FUNCTION_BLOCK FB_Tuer
VAR_INPUT
	SensorOpen1 : BOOL;
	SensorOpen2 : BOOL;
	SensorOpen3 : BOOL;
	SensorOpen4 : BOOL;
	SensorOpen5 : BOOL;
	SensorOpen6 : BOOL;
	
	SensorClosed1 : BOOL;
	SensorClosed2 : BOOL;
	SensorClosed3 : BOOL;
	SensorClosed4 : BOOL;
	SensorClosed5 : BOOL;
	SensorClosed6 : BOOL;
	
	Lichtschranke1 : BOOL;
	Lichtschranke2 : BOOL;
	Lichtschranke3 : BOOL;
	Lichtschranke4 : BOOL;
	Lichtschranke5 : BOOL;
	Lichtschranke6 : BOOL;
END_VAR
VAR_OUTPUT
	MotorOpen1 : BOOL;
	MotorOpen2 : BOOL;
	MotorOpen3 : BOOL;
	MotorOpen4 : BOOL;
	MotorOpen5 : BOOL;
	MotorOpen6 : BOOL;
	
	MotorClose1 : BOOL;
	MotorClose2 : BOOL;
	MotorClose3 : BOOL;
	MotorClose4 : BOOL;
	MotorClose5 : BOOL;
	MotorClose6 : BOOL;
	Done : BOOL;
	AllDoorsClosed : BOOL;
END_VAR
VAR
	TuerzyklusStarten : BOOL;
	Stockwerk : INT;
	State : ENUM_Tuer;
	ton1 : TON;
	ton2 : TON;
	ton3 : TON;
	ton4 : TON;
	ton5 : TON;
	ton6 : TON;
	Tueroffen : BOOL;
	bCloseAllMode : BOOL;
END_VAR

Done := FALSE;
ton1(IN := State = ENUM_Tuer.TuereAuf AND SensorOpen1, PT := T#2S);
ton2(IN := State = ENUM_Tuer.TuereAuf AND SensorOpen2, PT := T#2S);
ton3(IN := State = ENUM_Tuer.TuereAuf AND SensorOpen3, PT := T#2S);
ton4(IN := State = ENUM_Tuer.TuereAuf AND SensorOpen4, PT := T#2S);
ton5(IN := State = ENUM_Tuer.TuereAuf AND SensorOpen5, PT := T#2S);
ton6(IN := State = ENUM_Tuer.TuereAuf AND SensorOpen6, PT := T#2S);
IF bCloseAllMode THEN
    // Alle Türen schliessen – normaler State-Machine wird überbrückt
    MotorOpen1 := FALSE;
    IF NOT Lichtschranke1 THEN
        MotorClose1 := FALSE;
    ELSIF NOT SensorClosed1 THEN
        MotorClose1 := TRUE;
    ELSE
        MotorClose1 := FALSE;
    END_IF
    MotorOpen2 := FALSE;
    IF NOT Lichtschranke2 THEN
        MotorClose2 := FALSE;
    ELSIF NOT SensorClosed2 THEN
        MotorClose2 := TRUE;
    ELSE
        MotorClose2 := FALSE;
    END_IF
    MotorOpen3 := FALSE;
    IF NOT Lichtschranke3 THEN
        MotorClose3 := FALSE;
    ELSIF NOT SensorClosed3 THEN
        MotorClose3 := TRUE;
    ELSE
        MotorClose3 := FALSE;
    END_IF
    MotorOpen4 := FALSE;
    IF NOT Lichtschranke4 THEN
        MotorClose4 := FALSE;
    ELSIF NOT SensorClosed4 THEN
        MotorClose4 := TRUE;
    ELSE
        MotorClose4 := FALSE;
    END_IF
    MotorOpen5 := FALSE;
    IF NOT Lichtschranke5 THEN
        MotorClose5 := FALSE;
    ELSIF NOT SensorClosed5 THEN
        MotorClose5 := TRUE;
    ELSE
        MotorClose5 := FALSE;
    END_IF
    MotorOpen6 := FALSE;
    IF NOT Lichtschranke6 THEN
        MotorClose6 := FALSE;
    ELSIF NOT SensorClosed6 THEN
        MotorClose6 := TRUE;
    ELSE
        MotorClose6 := FALSE;
    END_IF
    // Wenn alle zu: Modus beenden
    IF SensorClosed1 AND SensorClosed2 AND SensorClosed3
       AND SensorClosed4 AND SensorClosed5 AND SensorClosed6 THEN
        bCloseAllMode := FALSE;
        Done := TRUE;
    END_IF
ELSE
    // Normaler Betrieb: Ausgänge zurücksetzen, dann State-Machine
    MotorOpen1 := FALSE;
    MotorClose1 := FALSE;
    MotorOpen2 := FALSE;
    MotorClose2 := FALSE;
    MotorOpen3 := FALSE;
    MotorClose3 := FALSE;
    MotorOpen4 := FALSE;
    MotorClose4 := FALSE;
    MotorOpen5 := FALSE;
    MotorClose5 := FALSE;
    MotorOpen6 := FALSE;
    MotorClose6 := FALSE;
    CASE State OF
        ENUM_Tuer.TuereZu:
            IF TuerzyklusStarten AND Stockwerk = 1 THEN
                State := ENUM_Tuer.TuereOeffnen;
            END_IF
            IF TuerzyklusStarten AND Stockwerk = 2 THEN
                State := ENUM_Tuer.TuereOeffnen;
            END_IF
            IF TuerzyklusStarten AND Stockwerk = 3 THEN
                State := ENUM_Tuer.TuereOeffnen;
            END_IF
            IF TuerzyklusStarten AND Stockwerk = 4 THEN
                State := ENUM_Tuer.TuereOeffnen;
            END_IF
            IF TuerzyklusStarten AND Stockwerk = 5 THEN
                State := ENUM_Tuer.TuereOeffnen;
            END_IF
            IF TuerzyklusStarten AND Stockwerk = 6 THEN
                State := ENUM_Tuer.TuereOeffnen;
            END_IF
        ENUM_Tuer.TuereOeffnen:
            Tueroffen := TRUE;
            IF Stockwerk = 1 THEN
                IF NOT SensorOpen1 THEN
                    MotorOpen1 := TRUE;
                ELSE
                    MotorOpen1 := FALSE;
                    State := ENUM_Tuer.TuereAuf;
                END_IF
            END_IF
            IF Stockwerk = 2 THEN
                IF NOT SensorOpen2 THEN
                    MotorOpen2 := TRUE;
                ELSE
                    MotorOpen2 := FALSE;
                    State := ENUM_Tuer.TuereAuf;
                END_IF
            END_IF
            IF Stockwerk = 3 THEN
                IF NOT SensorOpen3 THEN
                    MotorOpen3 := TRUE;
                ELSE
                    MotorOpen3 := FALSE;
                    State := ENUM_Tuer.TuereAuf;
                END_IF
            END_IF
            IF Stockwerk = 4 THEN
                IF NOT SensorOpen4 THEN
                    MotorOpen4 := TRUE;
                ELSE
                    MotorOpen4 := FALSE;
                    State := ENUM_Tuer.TuereAuf;
                END_IF
            END_IF
            IF Stockwerk = 5 THEN
                IF NOT SensorOpen5 THEN
                    MotorOpen5 := TRUE;
                ELSE
                    MotorOpen5 := FALSE;
                    State := ENUM_Tuer.TuereAuf;
                END_IF
            END_IF
            IF Stockwerk = 6 THEN
                IF NOT SensorOpen6 THEN
                    MotorOpen6 := TRUE;
                ELSE
                    MotorOpen6 := FALSE;
                    State := ENUM_Tuer.TuereAuf;
                END_IF
            END_IF
        ENUM_Tuer.TuereAuf:
            Tueroffen := FALSE;
            IF Stockwerk = 1 AND ton1.Q THEN
                State := ENUM_Tuer.TuereSchliessen;
            END_IF
            IF Stockwerk = 2 AND ton2.Q THEN
                State := ENUM_Tuer.TuereSchliessen;
            END_IF
            IF Stockwerk = 3 AND ton3.Q THEN
                State := ENUM_Tuer.TuereSchliessen;
            END_IF
            IF Stockwerk = 4 AND ton4.Q THEN
                State := ENUM_Tuer.TuereSchliessen;
            END_IF
            IF Stockwerk = 5 AND ton5.Q THEN
                State := ENUM_Tuer.TuereSchliessen;
            END_IF
            IF Stockwerk = 6 AND ton6.Q THEN
                State := ENUM_Tuer.TuereSchliessen;
            END_IF
        ENUM_Tuer.TuereSchliessen:
            IF Stockwerk = 1 THEN
                IF NOT Lichtschranke1 THEN
                    MotorClose1 := FALSE;
                    State := ENUM_Tuer.TuereOeffnen;
                ELSIF NOT SensorClosed1 THEN
                    MotorClose1 := TRUE;
                ELSE
                    MotorClose1 := FALSE;
                    TuerzyklusStarten := FALSE;
                    Done := TRUE;
                    State := ENUM_Tuer.TuereZu;
                END_IF
            END_IF
            IF Stockwerk = 2 THEN
                IF NOT Lichtschranke2 THEN
                    MotorClose2 := FALSE;
                    State := ENUM_Tuer.TuereOeffnen;
                ELSIF NOT SensorClosed2 THEN
                    MotorClose2 := TRUE;
                ELSE
                    MotorClose2 := FALSE;
                    TuerzyklusStarten := FALSE;
                    Done := TRUE;
                    State := ENUM_Tuer.TuereZu;
                END_IF
            END_IF
            IF Stockwerk = 3 THEN
                IF NOT Lichtschranke3 THEN
                    MotorClose3 := FALSE;
                    State := ENUM_Tuer.TuereOeffnen;
                ELSIF NOT SensorClosed3 THEN
                    MotorClose3 := TRUE;
                ELSE
                    MotorClose3 := FALSE;
                    TuerzyklusStarten := FALSE;
                    Done := TRUE;
                    State := ENUM_Tuer.TuereZu;
                END_IF
            END_IF
            IF Stockwerk = 4 THEN
                IF NOT Lichtschranke4 THEN
                    MotorClose4 := FALSE;
                    State := ENUM_Tuer.TuereOeffnen;
                ELSIF NOT SensorClosed4 THEN
                    MotorClose4 := TRUE;
                ELSE
                    MotorClose4 := FALSE;
                    TuerzyklusStarten := FALSE;
                    Done := TRUE;
                    State := ENUM_Tuer.TuereZu;
                END_IF
            END_IF
            IF Stockwerk = 5 THEN
                IF NOT Lichtschranke5 THEN
                    MotorClose5 := FALSE;
                    State := ENUM_Tuer.TuereOeffnen;
                ELSIF NOT SensorClosed5 THEN
                    MotorClose5 := TRUE;
                ELSE
                    MotorClose5 := FALSE;
                    TuerzyklusStarten := FALSE;
                    Done := TRUE;
                    State := ENUM_Tuer.TuereZu;
                END_IF
            END_IF
            IF Stockwerk = 6 THEN
                IF NOT Lichtschranke6 THEN
                    MotorClose6 := FALSE;
                    State := ENUM_Tuer.TuereOeffnen;
                ELSIF NOT SensorClosed6 THEN
                    MotorClose6 := TRUE;
                ELSE
                    MotorClose6 := FALSE;
                    TuerzyklusStarten := FALSE;
                    Done := TRUE;
                    State := ENUM_Tuer.TuereZu;
                END_IF
            END_IF
        ENUM_Tuer.Error:
    END_CASE
END_IF

IF IO_L1.Door_1_SensorClosed AND IO_L1.Door_2_SensorClosed AND IO_L1.Door_3_SensorClosed AND IO_L1.Door_4_SensorClosed AND IO_L1.Door_5_SensorClosed AND IO_L1.Door_6_SensorClosed THEN
	AllDoorsClosed := TRUE;
ELSE
	AllDoorsClosed := FALSE;
END_IF

METHOD PUBLIC M_AreDoorsClosed : BOOL
VAR_INPUT
END_VAR
IF IO_L1.Door_1_SensorClosed AND IO_L1.Door_2_SensorClosed AND IO_L1.Door_3_SensorClosed AND IO_L1.Door_4_SensorClosed AND IO_L1.Door_5_SensorClosed AND IO_L1.Door_6_SensorClosed THEN
	M_AreDoorsClosed := TRUE;
ELSE
	M_AreDoorsClosed := FALSE;
END_IF
END_METHOD

METHOD PUBLIC M_closeAllDoors : BOOL
VAR_INPUT
END_VAR
VAR
	Tuer1zu : BOOL;
	Tuer2zu : BOOL;
	Tuer3zu : BOOL;
	Tuer4zu : BOOL;
	Tuer5zu : BOOL;
	Tuer6zu : BOOL;
END_VAR

bCloseAllMode := TRUE;

M_closeAllDoors :=
    SensorClosed1 AND SensorClosed2 AND SensorClosed3 AND
    SensorClosed4 AND SensorClosed5 AND SensorClosed6;
END_METHOD

METHOD PUBLIC M_DoorOpen : BOOL
VAR_INPUT
	
END_VAR
IF Tueroffen THEN
	M_DoorOpen := TRUE;
ELSE
	M_DoorOpen := FALSE;
END_IF
END_METHOD

METHOD PUBLIC M_isDone : BOOL
VAR_INPUT
END_VAR
IF Done THEN
	M_isDone := TRUE;
ELSE 
	M_isDone := FALSE;
END_IF
END_METHOD

METHOD PUBLIC M_Tuerablaufstarten : BOOL
VAR_INPUT
	m_Stockwerk : INT;
END_VAR
IF m_Stockwerk >= 1 AND m_Stockwerk <= 6 THEN
	TuerzyklusStarten := TRUE;
	Stockwerk := m_Stockwerk;
	M_Tuerablaufstarten := TRUE;
ELSE
	M_Tuerablaufstarten := FALSE;
END_IF
END_METHOD

END_FUNCTION_BLOCK

(* stored: Version 1.1.0.1
   POU FB_Tuer: Id {ce7c9125-ad9c-4e95-8ddd-f81fee6abf98}, SpecialFunc None
   Method M_AreDoorsClosed: Id {b26a9bf4-2fc3-4358-ace3-7830ae6fabe9}
   Method M_closeAllDoors: Id {76e9d497-3022-48bc-94a5-209742ec32d4}
   Method M_DoorOpen: Id {a81e80dc-9065-490b-b6a8-8ed585863b63}
   Method M_isDone: Id {fc2b4786-e2ff-464a-9600-bf8dbab54ba4}
   Method M_Tuerablaufstarten: Id {51df235a-8b8a-4d18-9616-6b8239ca1c31} *)
